Fanuc KAREL source: kt00898.KL

-- PROVISIONAL review KL for V1013-1; original PC SHA256 7eee6174b700ed135e54fbc169c2b39c2b59381d3de2d874285b23dc9ec1ec92
-- Incomplete behavior may be omitted. Consult companion uncertainty JSON. Do not deploy.
PROGRAM KT00898
%NOLOCKGROUP
VAR
  OUT : BOOLEAN
-- UNRESOLVED_DECL P1 type=000101
-- UNRESOLVED_DECL P2 type=000101
BEGIN
  -- UNRESOLVED_PC offsets 5-31; opcodes 27,27,49,7E,AD,27,9D,76,23
  -- UNRESOLVED_PC offsets 36-40; opcodes 7F
END KT00898
